{attribute 'qualified_only'}
VAR_GLOBAL CONSTANT 
  uiNumIrrLinesForHMI_C         : UINT := 1;//how many robots are handled by a single PLC/HMI
  uiNumIrrLinesInGreenhouse_C   : UINT := 2;//2 Telegram BOT, one for each line or bay or span of the greenhouse, selected based on line number

  tTimeOutAxisMC_C              : TIME := T#3S;
  tTimeOutAxisMasterMC_C        : TIME := T#3S;
  uiRetryPowerOnCnt_C           : UINT := 6;
  
  lrAroundZero_C                : LREAL := 0.18; // m/s //used to check if velocity is around 0 m/s
END_VAR

(* stored: Version 1.1.0.1, ProductVersion 3.1.4024.12
   GVL C: Id {0308330d-e4af-4094-9b92-88c207c3c970} *)
